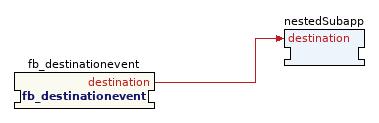
      [picture p25: application EventConnectionTestApp.Test8Solution]
      FBS
        fb_destinationevent : fb_destinationevent;
      END_FBS
      SUBAPPLICATION nestedSubapp
        EVENT_INPUT
          destination;
        END_EVENT
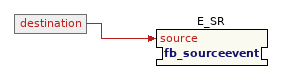
        FBS
          E_SR : fb_sourceevent;
        END_FBS
        EVENT_CONNECTIONS
          destination TO E_SR.source;
        END_CONNECTIONS
      END_SUBAPPLICATION
      EVENT_CONNECTIONS
        fb_destinationevent.destination TO nestedSubapp.destination;
      END_CONNECTIONS
    END_SUBAPPLICATION
    SUBAPPLICATION Test9 (* crossing connection from subapp interface to twice nested subapp via app network *)
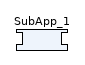
      SUBAPPLICATION SubApp_1
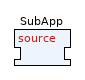
        SUBAPPLICATION SubApp
          EVENT_INPUT
            source;
          END_EVENT
        END_SUBAPPLICATION
      END_SUBAPPLICATION
    END_SUBAPPLICATION
    SUBAPPLICATION SubApp
      EVENT_OUTPUT
        destination;
      END_EVENT
    END_SUBAPPLICATION
    SUBAPPLICATION Test9Solution
      EVENT_INPUT
        destination;
      END_EVENT
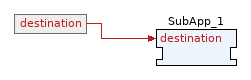
      SUBAPPLICATION SubApp_1
        EVENT_INPUT
          destination;
        END_EVENT
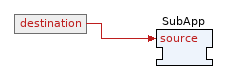
        SUBAPPLICATION SubApp
          EVENT_INPUT
            source;
          END_EVENT
        END_SUBAPPLICATION
        EVENT_CONNECTIONS
          destination TO SubApp.source;
        END_CONNECTIONS
      END_SUBAPPLICATION
      EVENT_CONNECTIONS
        destination TO SubApp_1.destination;
      END_CONNECTIONS
    END_SUBAPPLICATION
    SUBAPPLICATION SubApp_1
      EVENT_OUTPUT
        destination;
      END_EVENT
    END_SUBAPPLICATION
    SUBAPPLICATION Test10 (* crossing connection from subapp interface to twice nested subapp via app network *)
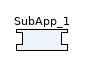
      SUBAPPLICATION SubApp_1
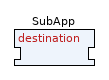
        SUBAPPLICATION SubApp
          EVENT_INPUT
            destination;
          END_EVENT
        END_SUBAPPLICATION
      END_SUBAPPLICATION
    END_SUBAPPLICATION
    SUBAPPLICATION SubApp_2
      EVENT_OUTPUT
        source;
      END_EVENT
    END_SUBAPPLICATION
    SUBAPPLICATION Test10Solution
      EVENT_INPUT
        source;
      END_EVENT
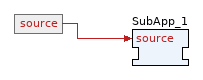
      SUBAPPLICATION SubApp_1
        EVENT_INPUT
          source;
        END_EVENT
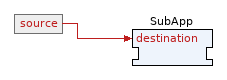
        SUBAPPLICATION SubApp
          EVENT_INPUT
            destination;
          END_EVENT
        END_SUBAPPLICATION
        EVENT_CONNECTIONS
          source TO SubApp.destination;
        END_CONNECTIONS
      END_SUBAPPLICATION
      EVENT_CONNECTIONS
        source TO SubApp_1.source;
      END_CONNECTIONS
    END_SUBAPPLICATION
    SUBAPPLICATION SubApp_3
      EVENT_OUTPUT
        source;
      END_EVENT
    END_SUBAPPLICATION
    SUBAPPLICATION Test11 (* crossing connection from subapp interface to twice nested subapp via app network + swap *)
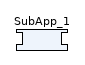
      SUBAPPLICATION SubApp_1
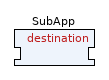
        SUBAPPLICATION SubApp
          EVENT_OUTPUT
            destination;
          END_EVENT
        END_SUBAPPLICATION
      END_SUBAPPLICATION
    END_SUBAPPLICATION
    SUBAPPLICATION SubApp_4
      EVENT_OUTPUT
        source;
      END_EVENT
    END_SUBAPPLICATION
    SUBAPPLICATION Test11Solution
      EVENT_INPUT
        source;
      END_EVENT
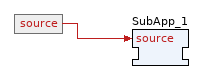
      SUBAPPLICATION SubApp_1
        EVENT_INPUT
          source;
        END_EVENT
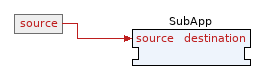
        SUBAPPLICATION SubApp
          EVENT_INPUT
            source;
          END_EVENT
          EVENT_OUTPUT
            destination;
          END_EVENT
          EVENT_CONNECTIONS
            source TO destination;
          END_CONNECTIONS
        END_SUBAPPLICATION
        EVENT_CONNECTIONS
          source TO SubApp.source;
        END_CONNECTIONS
      END_SUBAPPLICATION
      EVENT_CONNECTIONS
        source TO SubApp_1.source;
      END_CONNECTIONS
    END_SUBAPPLICATION
    SUBAPPLICATION SubApp_5
      EVENT_OUTPUT
        source;
      END_EVENT
    END_SUBAPPLICATION
    SUBAPPLICATION Test12 (* crossing connection from twice nested subapp to subapp interface via app network *)
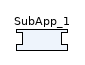
      SUBAPPLICATION SubApp_1
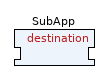
        SUBAPPLICATION SubApp
          EVENT_OUTPUT
            destination;
          END_EVENT
        END_SUBAPPLICATION
      END_SUBAPPLICATION
    END_SUBAPPLICATION
    SUBAPPLICATION SubApp_6
      EVENT_INPUT
        source;
      END_EVENT
    END_SUBAPPLICATION
    SUBAPPLICATION Test12Solution
      EVENT_OUTPUT
        destination;
      END_EVENT
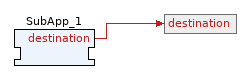
      SUBAPPLICATION SubApp_1
        EVENT_OUTPUT
          destination;
        END_EVENT
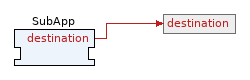
        SUBAPPLICATION SubApp
          EVENT_OUTPUT
            destination;
          END_EVENT
        END_SUBAPPLICATION
        EVENT_CONNECTIONS
          SubApp.destination TO destination;
        END_CONNECTIONS
      END_SUBAPPLICATION
      EVENT_CONNECTIONS
        SubApp_1.destination TO destination;
      END_CONNECTIONS
    END_SUBAPPLICATION
    SUBAPPLICATION SubApp_7
      EVENT_INPUT
        source;
      END_EVENT
    END_SUBAPPLICATION
    SUBAPPLICATION Test13 (* event input pin already exists outwards *)
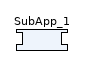
      SUBAPPLICATION SubApp_1
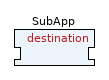
        SUBAPPLICATION SubApp
          EVENT_OUTPUT
            destination;
          END_EVENT
        END_SUBAPPLICATION
      END_SUBAPPLICATION
    END_SUBAPPLICATION
    SUBAPPLICATION SubApp_8
      EVENT_INPUT
        source;
      END_EVENT
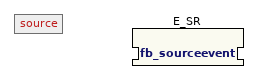
      FBS
        E_SR : fb_sourceevent;
      END_FBS
    END_SUBAPPLICATION
    SUBAPPLICATION Test13Solution
      EVENT_OUTPUT
        destination;
      END_EVENT
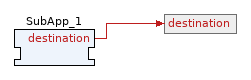
      SUBAPPLICATION SubApp_1
        EVENT_OUTPUT
          destination;
        END_EVENT
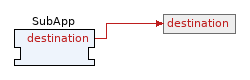
        SUBAPPLICATION SubApp
          EVENT_OUTPUT
            destination;
          END_EVENT
        END_SUBAPPLICATION
        EVENT_CONNECTIONS
          SubApp.destination TO destination;
        END_CONNECTIONS
      END_SUBAPPLICATION
      EVENT_CONNECTIONS
        SubApp_1.destination TO destination;
      END_CONNECTIONS
    END_SUBAPPLICATION
    SUBAPPLICATION SubApp_9
      EVENT_INPUT
        source;
      END_EVENT
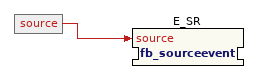
      FBS
        E_SR : fb_sourceevent;
      END_FBS
      EVENT_CONNECTIONS
        source TO E_SR.source;
      END_CONNECTIONS
    END_SUBAPPLICATION
    SUBAPPLICATION Test14 (* event input pin with same name already exists *)
